// TIA Portal V20 export
FUNCTION_BLOCK "Simulation"   // FB10, LAD
// stored: MemoryReserve 100, Namespace Unit1.Em4, SetENOAutomatically false
   VAR_INPUT
      simulation { ExternalAccessible := 'False'; ExternalVisible := 'False'; ExternalWritable := 'False'} : Bool;
   END_VAR
   VAR
      instMainPnPActuator { ExternalAccessible := 'False'; ExternalVisible := 'False'; ExternalWritable := 'False'} : Array[0..9] of "LER_SimActuator";
      instAlignTableActuator { ExternalAccessible := 'False'; ExternalVisible := 'False'; ExternalWritable := 'False'} : Array[0..9] of "LER_SimActuator";
      instNgPnPActuator { ExternalAccessible := 'False'; ExternalVisible := 'False'; ExternalWritable := 'False'} : Array[0..9] of "LER_SimActuator";
   END_VAR
   VAR_TEMP   // added for the SCL form of the ladder/FBD networks
      _w1 : Bool;
   END_VAR
BEGIN

REGION Network 1: Main P&P Two Way Actuator
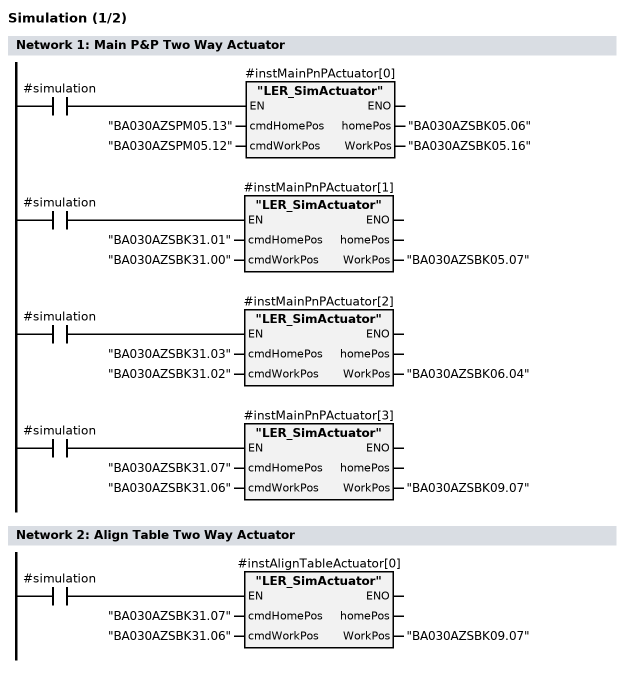
   RUNG wire#powerrail
      Contact( #simulation )
      #instMainPnPActuator[0](cmdHomePos := "BA030AZSPM05.13", cmdWorkPos := "BA030AZSPM05.12", homePos => "BA030AZSBK05.06", WorkPos => "BA030AZSBK05.16")
   END_RUNG
   RUNG wire#powerrail
      Contact( #simulation )
      #instMainPnPActuator[1](cmdHomePos := "BA030AZSBK31.01", cmdWorkPos := "BA030AZSBK31.00", homePos =>, WorkPos => "BA030AZSBK05.07")
   END_RUNG
   RUNG wire#powerrail
      Contact( #simulation )
      #instMainPnPActuator[2](cmdHomePos := "BA030AZSBK31.03", cmdWorkPos := "BA030AZSBK31.02", homePos =>, WorkPos => "BA030AZSBK06.04")
   END_RUNG
   RUNG wire#powerrail
      Contact( #simulation )
      #instMainPnPActuator[3](cmdHomePos := "BA030AZSBK31.07", cmdWorkPos := "BA030AZSBK31.06", homePos =>, WorkPos => "BA030AZSBK09.07")
   END_RUNG
   // the same network as SCL:
   IF #simulation THEN
       #instMainPnPActuator[0](cmdHomePos := "BA030AZSPM05.13",   // "LER_SimActuator"
                               cmdWorkPos := "BA030AZSPM05.12",
                               homePos => "BA030AZSBK05.06",
                               WorkPos => "BA030AZSBK05.16");
       #instMainPnPActuator[1](cmdHomePos := "BA030AZSBK31.01",   // "LER_SimActuator"
                               cmdWorkPos := "BA030AZSBK31.00",
                               WorkPos => "BA030AZSBK05.07");
       #instMainPnPActuator[2](cmdHomePos := "BA030AZSBK31.03",   // "LER_SimActuator"
                               cmdWorkPos := "BA030AZSBK31.02",
                               WorkPos => "BA030AZSBK06.04");
       #instMainPnPActuator[3](cmdHomePos := "BA030AZSBK31.07",   // "LER_SimActuator"
                               cmdWorkPos := "BA030AZSBK31.06",
                               WorkPos => "BA030AZSBK09.07");
   END_IF;
END_REGION

REGION Network 2: Align Table Two Way Actuator
   RUNG wire#powerrail
      Contact( #simulation )
      #instAlignTableActuator[0](cmdHomePos := "BA030AZSBK31.07", cmdWorkPos := "BA030AZSBK31.06", homePos =>, WorkPos => "BA030AZSBK09.07")
   END_RUNG
   // the same network as SCL:
   IF #simulation THEN
       #instAlignTableActuator[0](cmdHomePos := "BA030AZSBK31.07",   // "LER_SimActuator"
                               cmdWorkPos := "BA030AZSBK31.06",
                               WorkPos => "BA030AZSBK09.07");
   END_IF;
END_REGION

REGION Network 3: NG P&P Two Way Actuator
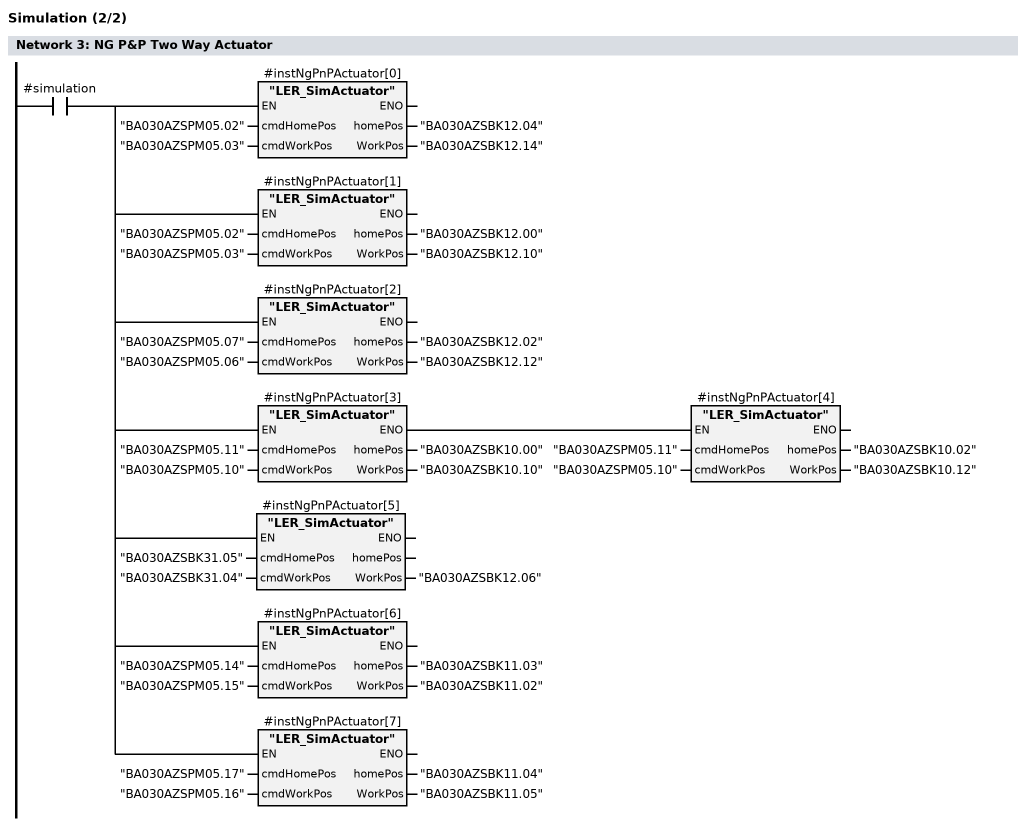
   RUNG wire#powerrail
      Contact( #simulation )
      wire#w1
      #instNgPnPActuator[0](cmdHomePos := "BA030AZSPM05.02", cmdWorkPos := "BA030AZSPM05.03", homePos => "BA030AZSBK12.04", WorkPos => "BA030AZSBK12.14")
   END_RUNG
   RUNG wire#w1
      #instNgPnPActuator[1](cmdHomePos := "BA030AZSPM05.02", cmdWorkPos := "BA030AZSPM05.03", homePos => "BA030AZSBK12.00", WorkPos => "BA030AZSBK12.10")
   END_RUNG
   RUNG wire#w1
      #instNgPnPActuator[2](cmdHomePos := "BA030AZSPM05.07", cmdWorkPos := "BA030AZSPM05.06", homePos => "BA030AZSBK12.02", WorkPos => "BA030AZSBK12.12")
   END_RUNG
   RUNG wire#w1
      #instNgPnPActuator[3](cmdHomePos := "BA030AZSPM05.11", cmdWorkPos := "BA030AZSPM05.10", homePos => "BA030AZSBK10.00", WorkPos => "BA030AZSBK10.10")
      #instNgPnPActuator[4](cmdHomePos := "BA030AZSPM05.11", cmdWorkPos := "BA030AZSPM05.10", homePos => "BA030AZSBK10.02", WorkPos => "BA030AZSBK10.12")
   END_RUNG
   RUNG wire#w1
      #instNgPnPActuator[5](cmdHomePos := "BA030AZSBK31.05", cmdWorkPos := "BA030AZSBK31.04", homePos =>, WorkPos => "BA030AZSBK12.06")
   END_RUNG
   RUNG wire#w1
      #instNgPnPActuator[6](cmdHomePos := "BA030AZSPM05.14", cmdWorkPos := "BA030AZSPM05.15", homePos => "BA030AZSBK11.03", WorkPos => "BA030AZSBK11.02")
   END_RUNG
   RUNG wire#w1
      #instNgPnPActuator[7](cmdHomePos := "BA030AZSPM05.17", cmdWorkPos := "BA030AZSPM05.16", homePos => "BA030AZSBK11.04", WorkPos => "BA030AZSBK11.05")
   END_RUNG
   // the same network as SCL:
   IF #simulation THEN
       #instNgPnPActuator[0](cmdHomePos := "BA030AZSPM05.02",   // "LER_SimActuator"
                             cmdWorkPos := "BA030AZSPM05.03",
                             homePos => "BA030AZSBK12.04",
                             WorkPos => "BA030AZSBK12.14");
       #instNgPnPActuator[1](cmdHomePos := "BA030AZSPM05.02",   // "LER_SimActuator"
                             cmdWorkPos := "BA030AZSPM05.03",
                             homePos => "BA030AZSBK12.00",
                             WorkPos => "BA030AZSBK12.10");
       #instNgPnPActuator[2](cmdHomePos := "BA030AZSPM05.07",   // "LER_SimActuator"
                             cmdWorkPos := "BA030AZSPM05.06",
                             homePos => "BA030AZSBK12.02",
                             WorkPos => "BA030AZSBK12.12");
   END_IF;
   #instNgPnPActuator[3](EN := #simulation,   // "LER_SimActuator"
                         cmdHomePos := "BA030AZSPM05.11",
                         cmdWorkPos := "BA030AZSPM05.10",
                         homePos => "BA030AZSBK10.00",
                         WorkPos => "BA030AZSBK10.10",
                         ENO => #_w1);
   IF #_w1 THEN
       #instNgPnPActuator[4](cmdHomePos := "BA030AZSPM05.11",   // "LER_SimActuator"
                             cmdWorkPos := "BA030AZSPM05.10",
                             homePos => "BA030AZSBK10.02",
                             WorkPos => "BA030AZSBK10.12");
   END_IF;
   IF #simulation THEN
       #instNgPnPActuator[5](cmdHomePos := "BA030AZSBK31.05",   // "LER_SimActuator"
                             cmdWorkPos := "BA030AZSBK31.04",
                             WorkPos => "BA030AZSBK12.06");
       #instNgPnPActuator[6](cmdHomePos := "BA030AZSPM05.14",   // "LER_SimActuator"
                             cmdWorkPos := "BA030AZSPM05.15",
                             homePos => "BA030AZSBK11.03",
                             WorkPos => "BA030AZSBK11.02");
       #instNgPnPActuator[7](cmdHomePos := "BA030AZSPM05.17",   // "LER_SimActuator"
                             cmdWorkPos := "BA030AZSPM05.16",
                             homePos => "BA030AZSBK11.04",
                             WorkPos => "BA030AZSBK11.05");
   END_IF;
END_REGION
END_FUNCTION_BLOCK
